(* CODESYS project WagoAppCloud_MqttPubSub_Test_1.ecp
   Company: WAGO
   Title: WagoAppCloud_CostumerProtocol
   Description: Example for the Cloud Conectivity using MQTT with the own customer data strucure
   Author: wago / u014791
   Version: 1.0.0.0

Project tree, tasks and I/O mapping:
  PFC : 750-8212 PFC200 2ETH RS, WAGO, order no. 0750-8212, version 5.13.2.22
    application Application
      libraries: WagoAppString, 1.6.3.0 (WAGO); WagoAppCloud, * (WAGO); WagoAppConfigTool, 1.1.2.0 (WAGO)
      task Task (cyclic, interval t#10ms, priority 14) calls PLC_PRG
      program Status_NativeMQTT [ST]
      program Publish_NativeMQTT [ST]
      program PLC_PRG [ST]
      program Subscribe_NativeMQTT [ST]
    Kbus : Kbus, WAGO, version 1.4.0.2
        unmapped channels: K-BUS diagnostics
    MODBUS
      MODBUS : MODBUS, WAGO, order no. n/a, version 1.1.1.15
        LocalDeviceModbus : MODBUS Slave, WAGO, order no. n/a, version 1.1.1.15
            settings: OffsetMap = 0
            input  MbMqttTopicPart : WORD  // 
          TcpSettings : Modbus TCP Slave, WAGO, order no. n/a, version 1.1.1.15
              settings: TCP connection watchdog = 200 10ms
    Serial
      COM1 : COM1, WAGO, version 0.0.0.19
    Common.PCI
  Generic_MODBUS_Master : ThirdParty Modbus Master, WAGO, order no. GenericModbusMaster, version 1.0.0.1
*)

// PFC/Application/PLC_PRG
PROGRAM PLC_PRG
VAR

END_VAR


Publish_NativeMQTT();
Subscribe_NativeMQTT();
Status_NativeMQTT();

END_PROGRAM

// PFC/Application/Publish_NativeMQTT
// !!! IMPORTANT !!!
// Some cloud platforms have limitations on their MQTT-Implementation.
// Typically the supported payload size is significantly less then told by MQTT-Specification:
// it is 128KB for IBM Bluemix and Amazon Web Services (https://docs.aws.amazon.com/iot/latest/developerguide/protocols.html)
// Other known limitations are related to Quality Of Service Level, Retain message flag, ...
// !!! IMPORTANT !!!

// Purpose of the example program: Primitive JSON document shall periodically be published via dataagent daemon

PROGRAM Publish_NativeMQTT
VAR
	MyInterval		: TIME := T#5S;
	Timer			: TON;
	
	dwMyCounter 	: DWORD := 1;
	MyString 		: STRING(255);
	aBuffer			: ARRAY[0..255] OF BYTE;
	dwBytesCount 	: DWORD;
	
	oFbPublish 		: WagoAppCloud.FbPublishMQTT;
	xMyTrigger		: BOOL := FALSE;
	dwBusyCounter	: DWORD := 0;
	dwErrorCounter	: DWORD := 0;
	sTopic: STRING(255) := 'v1/devices/me/telemetry';
END_VAR

dwMyCounter := dwMyCounter + 1;

Timer(IN := TRUE, PT := MyInterval);
IF Timer.Q THEN
	Timer(IN := FALSE);

	IF NOT oFbPublish.xBusy THEN
		// Write primitive JSON into string (use WagoAppJson library for advanced JSON functionalities)
		MyString := CONCAT('{"MyCounter":', DWORD_TO_STRING(dwMyCounter));
		MyString := CONCAT(MyString, '}');
		// Copy JSON to buffer
		dwBytesCount := Length(MyString);
		MemCopy(pDest := ADR(aBuffer), pSource := ADR(MyString), udiSize := dwBytesCount);
		// Trigger the transmission
		xMyTrigger := TRUE;
	ELSE
		// Busy statistics counter
		dwBusyCounter := dwBusyCounter + 1;
	END_IF
	
	IF oFbPublish.xError THEN
		// Error statistics counter
		dwErrorCounter := dwErrorCounter + 1;
	END_IF
	
END_IF

// Trigger MQTT publish
oFbPublish(sTopic := sTopic,
			eQualityOfService := 1,
			dwSize := dwBytesCount,
			aData := aBuffer,
			xTrigger := xMyTrigger);

END_PROGRAM

// PFC/Application/Subscribe_NativeMQTT
PROGRAM Subscribe_NativeMQTT
VAR
	dwCycleCount		: DWORD := 0;	

	oFbSubscribe1 		: WagoAppCloud.FbSubscribeMQTT;
	aSubscriptionData1	: ARRAY [0..254] OF BYTE;
	sMessage1			: STRING(255);
	
	oFbSubscribe2 		: WagoAppCloud.FbSubscribeMQTT;
	aSubscriptionData2	: ARRAY [0..254] OF BYTE;
	sMessage2			: STRING(255);
	sSubscriptionData2: POINTER TO BYTE;
	sTopic: STRING(255) := 'v1/devices/me/telemetry';
END_VAR


dwCycleCount := dwCycleCount + 1;

IoConfig_Globals_Mapping.MbMqttTopicPart;

(*oFbSubscribe1(xSubscribe := TRUE, sTopic := 'MyTopic1', eQoS := eQualityOfService.QoS1, aPayloadData:= aSubscriptionData1);*)
oFbSubscribe1(xSubscribe := TRUE, sTopic := sTopic, eQoS := eQualityOfService.QoS1, aPayloadData:= aSubscriptionData1);
MemCopySecure(pDest:= ADR(sMessage1), udiDestSize:= 255, pSource:= ADR(aSubscriptionData1), udiSourceSize:= oFbSubscribe1.dwRxNBytes, bPadding:= 0);
(*
oFbSubscribe2(xSubscribe := TRUE, sTopic := 'MyTopic2', eQoS := eQualityOfService.QoS1, aPayloadData:= aSubscriptionData2);
MemCopySecure(pDest:= ADR(sMessage2), udiDestSize:= 255, pSource:= ADR(aSubscriptionData2), udiSourceSize:= oFbSubscribe2.dwRxNBytes, bPadding:= 0);
*)

END_PROGRAM

// PFC/Application/Status_NativeMQTT
// Purpose of the example program: Check status of Native MQTT
PROGRAM Status_NativeMQTT
VAR
	oFbStatus 			: WagoAppCloud.FbStatus_NativeMQTT;
	xMyError			: BOOL := FALSE;
	xConnectedToMyCloud	: BOOL := FALSE;
	rMyFillLevel		: REAL := 0;
	uliMyOutgoingBlocks	: ULINT := 0;
END_VAR

// Will detect new values every 5 seconds
oFbStatus(xEnabled := TRUE,
		   xError => xMyError,
		   xCloudConnected => xConnectedToMyCloud,			// Will be FALSE after network timeout occured 
		   rCacheFillLevel => rMyFillLevel,					// Increasing value indicates bad network or overload
		   uliOutgoingDataBlocks => uliMyOutgoingBlocks);  	// Only for QoS 1 and 2. Increasing value indicates bad network or overload

END_PROGRAM
